(* PLC project Unnamed, Unknown Unnamed 1 *)
(* stored: creationDateTime 2023-03-29T00:03:16, modificationDateTime 2023-04-16T13:55:39 *)

PROGRAM Master_Program
  VAR
    Panel_Mag_Sensor AT %IX0.0 : BOOL;  (* Physcial Inputs on the Right Demostration Panel offset 4 input *)
    Panel_IR_Sensor AT %IX0.1 : BOOL;  (* Physcial Inputs on the Right Demostration Panel offset 6 input *)
    Panel_Motion_Sensor AT %IX0.2 : BOOL;  (* Physcial Inputs on the Right Demostration Panel offset 5 input *)
    Panel_GD_Remote_UP_PB AT %IX0.3 : BOOL;  (* Physcial Inputs on the Right Demostration Panel offset 7 input *)
    Panel_GD_Remote_DOWN_PB AT %IX0.4 : BOOL;  (* Physcial Inputs on the Right Demostration Panel offset 8 input *)
    Panel_FD_Lock_Signal AT %IX0.5 : BOOL;  (* Physcial Inputs on the Right Demostration Panel offset 9 input *)
    Panel_Arm_Panel_PB AT %IX0.6 : BOOL;  (* Physcial Inputs on the Right Demostration Panel offset 2 input *)
    Panel_Arm_House_PB AT %IX0.7 : BOOL;  (* Physcial Inputs on the Right Demostration Panel offset 3 input *)
    Panel_Reset_PB AT %IX1.0 : BOOL;  (* Physcial Inputs on the Right Demostration Panel offset 11 input *)
    Panel_FD_Unlock_Signal AT %IX1.1 : BOOL;  (* Physcial Inputs on the Right Demostration Panel offset 10 input *)
    Panel_Alarm_Light AT %QX0.0 : BOOL;  (* Alarm flashes when triggered offset 0 coil "Changed from 0.0 for testing" 102.3 for uno pin 13 *)
    Home_GD_Postion_Switch AT %IX102.0 : BOOL;  (* Physcial Inputs in the House Model offset 801 input *)
    Home_Mag_Sensor AT %IX102.1 : BOOL;  (* Physcial Inputs in the House Model offset 802 input *)
    Home_Motion_Sensor AT %IX102.2 : BOOL;  (* Physcial Inputs in the House Model offset 803 input *)
    Home_IR_Sensor AT %IX102.3 : BOOL;  (* Physcial Inputs in the House Model offset 804 input *)
    Home_Green_PB_Floor_01 AT %IX102.4 : BOOL;  (* Physcial Inputs in the House Model offset 805 input *)
    Home_Green_PB_Floor_02 AT %IX102.5 : BOOL;  (* Physcial Inputs in the House Model offset 806 input *)
    Home_Blue_PB_Floor_03 AT %IX102.6 : BOOL;  (* Physcial Inputs in the House Model offset 807 input *)
    Home_Red_PB_Floor_03 AT %IX102.7 : BOOL;  (* Physcial Inputs in the House Model offset 807 input *)
    Home_Green_LED_Floor_01 AT %QX100.0 : BOOL;  (* Digital output to control GD Motor offset 800 coil "Changed from 100.0 for testing" *)
    Home_Green_LED_Floor_02 AT %QX100.1 : BOOL;  (* Digital output to control GD Motor offset 801 coil *)
    Home_Green_LED_Floor_03 AT %QX100.2 : BOOL;  (* Digital output to control GD Motor offset 802 coil *)
    Home_White_LED_Floor_01 AT %QX100.3 : BOOL;  (* Digital output to control GD Motor offset 803 coil *)
    Home_White_LED_Floor_02 AT %QX100.4 : BOOL;  (* Digital output to control GD Motor offset 804 coil *)
    Home_White_LED_Floor_03 AT %QX100.5 : BOOL;  (* Digital output to control GD Motor offset 805 coil *)
    Home_White_LED_Floor_Backside AT %QX100.6 : BOOL;  (* Digital output to control GD Motor offset 806 coil *)
    Home_GD_Motor_UP AT %QX100.7 : BOOL;  (* Digital output to control GD Motor offset 807 coil *)
    Home_GD_Motor_DOWN AT %QX101.0 : BOOL;  (* Digital output to control GD Motor offset 808 coil *)
    Home_FD_Deadbolt AT %QX101.1 : BOOL;  (* Digital output to control FD Solenoid offset 809 coil *)
    Home_GD_Position AT %QX101.2 : BOOL;  (* Digital output to control GD Motor offset 810 coil *)
    Panel_Arm_Virtual_PB AT %QX10.0 : BOOL;  (* Virutal Push Button for HMI and attacks offset 80 coil *)
    Panel_Arm_Mag_Sensor_Virtual AT %QX10.1 : BOOL;  (* Virutal Push Button for HMI and attacks offset 81 coil *)
    Panel_Arm_Motion_Sensor_Virtual AT %QX10.2 : BOOL;  (* Virutal Push Button for HMI and attacks offset 82 coil *)
    Panel_Arm_IR_Sensor_Virtual AT %QX10.3 : BOOL;  (* Virutal Push Button for HMI and attacks offset 83 coil *)
    Panel_Mag_Sensor_Virtual AT %QX10.4 : BOOL;  (* Virutal Push Button for HMI and attacks offset 84 coil *)
    Panel_Motion_Sensor_Virtual AT %QX10.5 : BOOL;  (* Virutal Push Button for HMI and attacks offset 85 coil *)
    Panel_IR_Sensor_Virtual AT %QX10.6 : BOOL;  (* Virutal Push Button for HMI and attacks offset 86 coil *)
    Panel_GD_Up_OnOff_Virtual_PB AT %QX10.7 : BOOL;  (* Virutal Push Button for HMI and attacks offset 87 coil *)
    Panel_GD_Remote_Up_Virtual AT %QX11.0 : BOOL;  (* Virutal Push Button for HMI and attacks offset 88 coil *)
    Panel_GD_Down_OnOff_Virtual_PB AT %QX11.1 : BOOL;  (* Virutal Push Button for HMI and attacks offset 89 coil *)
    Panel_GD_Remote_Down_Virtual AT %QX11.2 : BOOL;  (* Virutal Push Button for HMI and attacks offset 90 coil *)
    Panel_FD_Lock_OnOff_Virtual_PB AT %QX11.3 : BOOL;  (* Virutal Push Button for HMI and attacks offset 91 coil *)
    Panel_FD_Lock_Signal_Virtual AT %QX11.4 : BOOL;  (* Virutal Push Button for HMI and attacks offset 92 coil *)
    Panel_FD_Unlock_OnOff_Virtual_PB AT %QX11.5 : BOOL;  (* Virutal Push Button for HMI and attacks offset 93 coil *)
    Panel_FD_Unlock_Signal_Virtual AT %QX11.6 : BOOL;  (* Virutal Push Button for HMI and attacks offset 94 coil *)
    Home_FD_Lock_Signal_Virtual AT %QX110.0 : BOOL;  (* Virutal Push Button for HMI and attacks offset 880 coil *)
    Home_FD_Unlock_Signal_Virtual AT %QX110.1 : BOOL;  (* Virutal Push Button for HMI and attacks offset 881 coil *)
    Home_Arm_Virtual_PB AT %QX110.2 : BOOL;  (* Virutal Push Button for HMI and attacks offset 882 coil *)
    Home_Arm_Mag_Sensor_Virtual AT %QX110.3 : BOOL;  (* Virutal Push Button for HMI and attacks offset 883 coil *)
    Home_Mag_Sensor_Virtual AT %QX110.4 : BOOL;  (* Virutal Push Button for HMI and attacks offset 884 coil *)
    Home_Arm_Motion_Sensor_Virtual AT %QX110.5 : BOOL;  (* Virutal Push Button for HMI and attacks offset 885 coil *)
    Home_Motion_Sensor_Virtual AT %QX110.6 : BOOL;  (* Virutal Push Button for HMI and attacks offset 886 coil *)
    Home_Arm_IR_Sensor_Virtual AT %QX110.7 : BOOL;  (* Virutal Push Button for HMI and attacks offset 887 coil *)
    Home_IR_Sensor_Virtual AT %QX111.0 : BOOL;  (* Virutal Push Button for HMI and attacks offset 888 coil *)
    Home_Green_PB_Auto_01 AT %QX111.2 : BOOL;  (* Virutal Push Button for HMI and attacks offset 890 coil *)
    Home_Green_PB_Auto_02 AT %QX111.4 : BOOL;  (* Virutal Push Button for HMI and attacks offset 892 coil *)
    Home_Green_PB_Auto_03 AT %QX111.6 : BOOL;  (* Virutal Push Button for HMI and attacks offset 894 coil *)
    Home_Green_LED_Reset_PB AT %QX111.7 : BOOL;  (* Virutal Push Button for HMI and attacks offset 895 coil *)
    Reset_Green_Lights AT %QX112.0 : BOOL;  (* Virutal Push Button for HMI and attacks offset 896 coil *)
  END_VAR
  VAR
    TON0 : TON;  (* Waits set number of seconds before reseting the green lights. *)
  END_VAR
  VAR
    Home_White_PD_Floor_01 AT %QX112.1 : BOOL;  (* Virutal Push Button for HMI and attacks offset 897 coil *)
    Home_White_PD_Floor_02 AT %QX112.2 : BOOL;  (* Virutal Push Button for HMI and attacks offset 898 coil *)
    Home_White_PD_Floor_03 AT %QX112.3 : BOOL;  (* Virutal Push Button for HMI and attacks offset 899 coil *)
    Home_White_PD_Backside AT %QX112.4 : BOOL;  (* Virutal Push Button for HMI and attacks offset 900 *)
    Home_Reset_PB_Virtual AT %QX112.5 : BOOL;  (* Virutal Push Button for HMI and attacks offset 901 *)
    Home_GD_OpenClose_Switch_Vir AT %QX112.6 : BOOL;  (* Virutal Push Button for HMI and attacks offset 902 "Testing" *)
  END_VAR

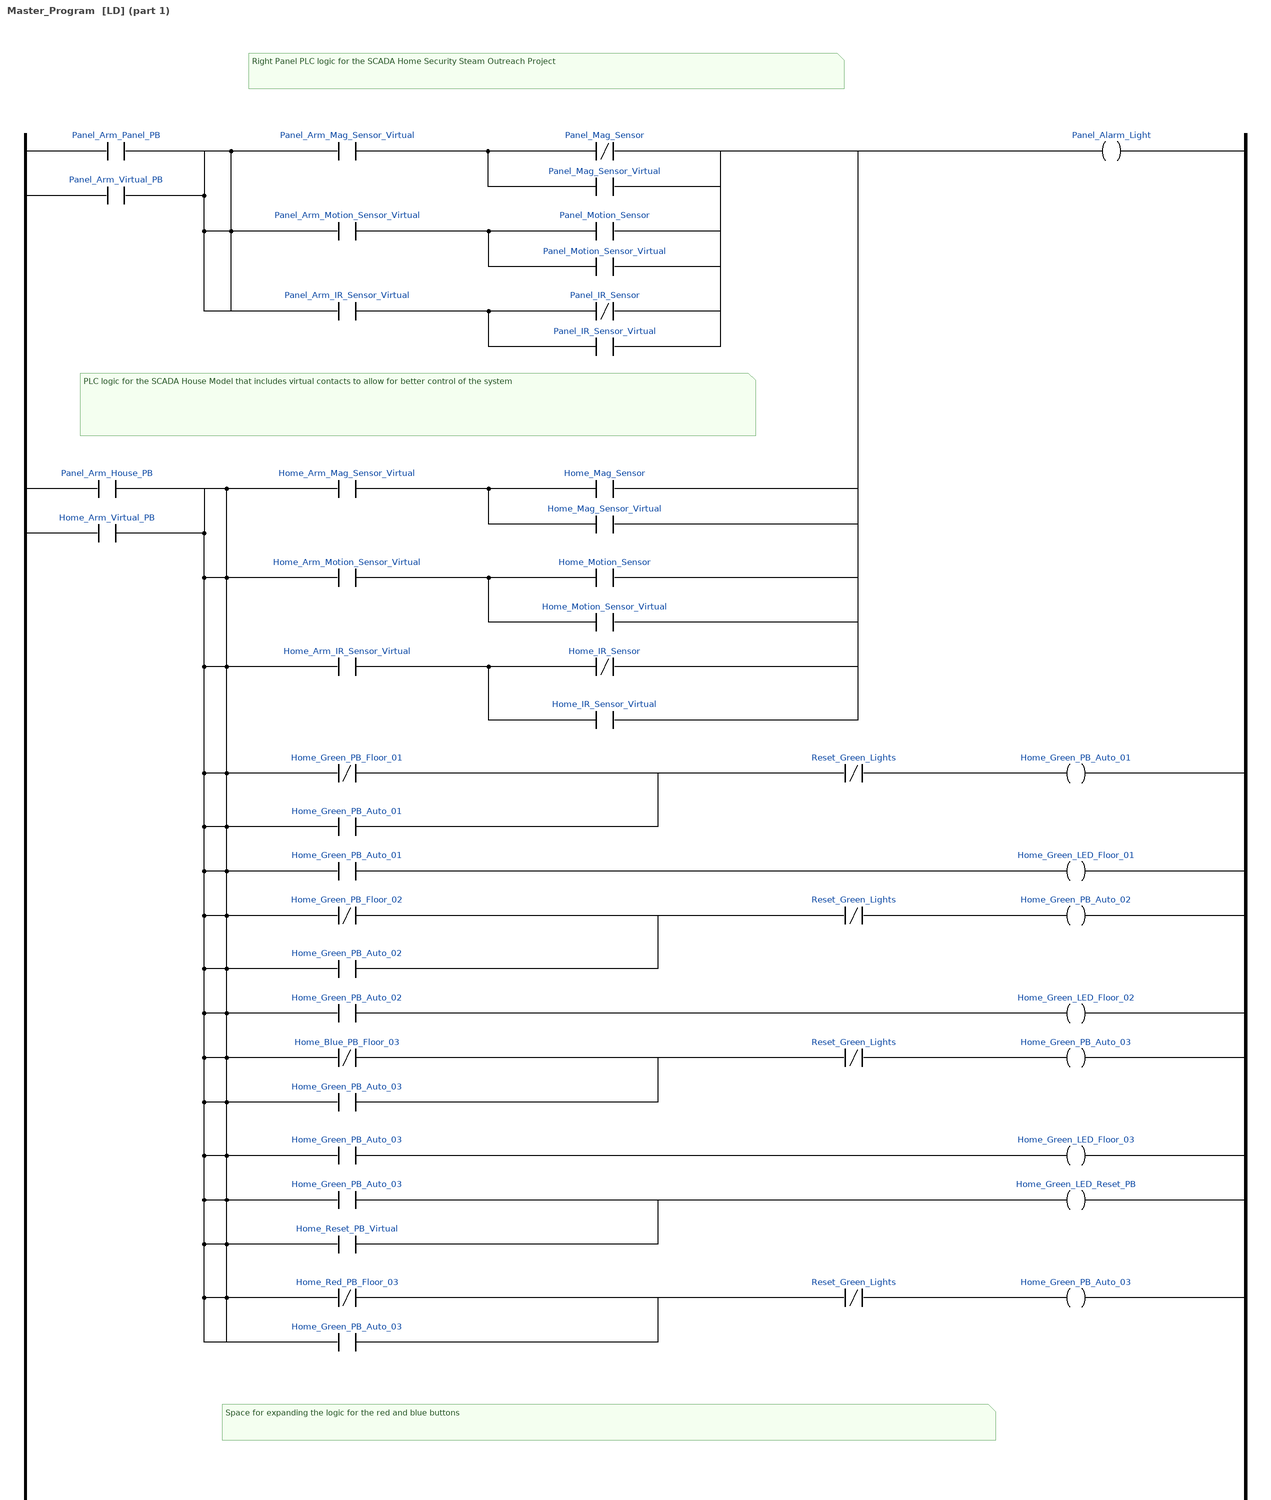
(* LD diagram, written out as Structured Text *)
(* Right Panel PLC logic for the SCADA Home Security Steam Outreach Project *)
Panel_Alarm_Light := (Panel_Arm_Panel_PB OR Panel_Arm_Virtual_PB) AND Panel_Arm_Mag_Sensor_Virtual AND NOT Panel_Mag_Sensor OR (Panel_Arm_Panel_PB OR Panel_Arm_Virtual_PB) AND Panel_Arm_Mag_Sensor_Virtual AND Panel_Mag_Sensor_Virtual OR (Panel_Arm_Panel_PB OR Panel_Arm_Virtual_PB) AND Panel_Arm_Motion_Sensor_Virtual AND Panel_Motion_Sensor OR (Panel_Arm_Panel_PB OR Panel_Arm_Virtual_PB) AND Panel_Arm_Motion_Sensor_Virtual AND Panel_Motion_Sensor_Virtual OR (Panel_Arm_Panel_PB OR Panel_Arm_Virtual_PB) AND Panel_Arm_IR_Sensor_Virtual AND NOT Panel_IR_Sensor OR (Panel_Arm_Panel_PB OR Panel_Arm_Virtual_PB) AND Panel_Arm_IR_Sensor_Virtual AND Panel_IR_Sensor_Virtual OR (Home_Arm_Virtual_PB OR Panel_Arm_House_PB) AND Home_Arm_Mag_Sensor_Virtual AND Home_Mag_Sensor OR (Home_Arm_Virtual_PB OR Panel_Arm_House_PB) AND Home_Arm_Mag_Sensor_Virtual AND Home_Mag_Sensor_Virtual OR (Home_Arm_Virtual_PB OR Panel_Arm_House_PB) AND Home_Arm_Motion_Sensor_Virtual AND Home_Motion_Sensor OR (Home_Arm_Virtual_PB OR Panel_Arm_House_PB) AND Home_Arm_Motion_Sensor_Virtual AND Home_Motion_Sensor_Virtual OR (Home_Arm_Virtual_PB OR Panel_Arm_House_PB) AND Home_Arm_IR_Sensor_Virtual AND NOT Home_IR_Sensor OR (Home_Arm_Virtual_PB OR Panel_Arm_House_PB) AND Home_Arm_IR_Sensor_Virtual AND Home_IR_Sensor_Virtual;
(* PLC logic for the SCADA House Model that includes virtual contacts to allow for better control of the system *)
Home_Green_PB_Auto_01 := (Panel_Arm_House_PB OR Home_Arm_Virtual_PB) AND (Home_Green_PB_Auto_01 OR NOT Home_Green_PB_Floor_01) AND NOT Reset_Green_Lights;
Home_Green_LED_Floor_01 := (Panel_Arm_House_PB OR Home_Arm_Virtual_PB) AND Home_Green_PB_Auto_01;
Home_Green_PB_Auto_02 := (Home_Arm_Virtual_PB OR Panel_Arm_House_PB) AND (Home_Green_PB_Auto_02 OR NOT Home_Green_PB_Floor_02) AND NOT Reset_Green_Lights;
Home_Green_LED_Floor_02 := (Home_Arm_Virtual_PB OR Panel_Arm_House_PB) AND Home_Green_PB_Auto_02;
Home_Green_PB_Auto_03 := (Home_Arm_Virtual_PB OR Panel_Arm_House_PB) AND (Home_Green_PB_Auto_03 OR NOT Home_Blue_PB_Floor_03) AND NOT Reset_Green_Lights;
Home_Green_LED_Floor_03 := (Home_Arm_Virtual_PB OR Panel_Arm_House_PB) AND Home_Green_PB_Auto_03;
Home_Green_LED_Reset_PB := (Home_Arm_Virtual_PB OR Panel_Arm_House_PB) AND (Home_Green_PB_Auto_03 OR Home_Reset_PB_Virtual);
Home_Green_PB_Auto_03 := (Panel_Arm_House_PB OR Home_Arm_Virtual_PB) AND (NOT Home_Red_PB_Floor_03 OR Home_Green_PB_Auto_03) AND NOT Reset_Green_Lights;
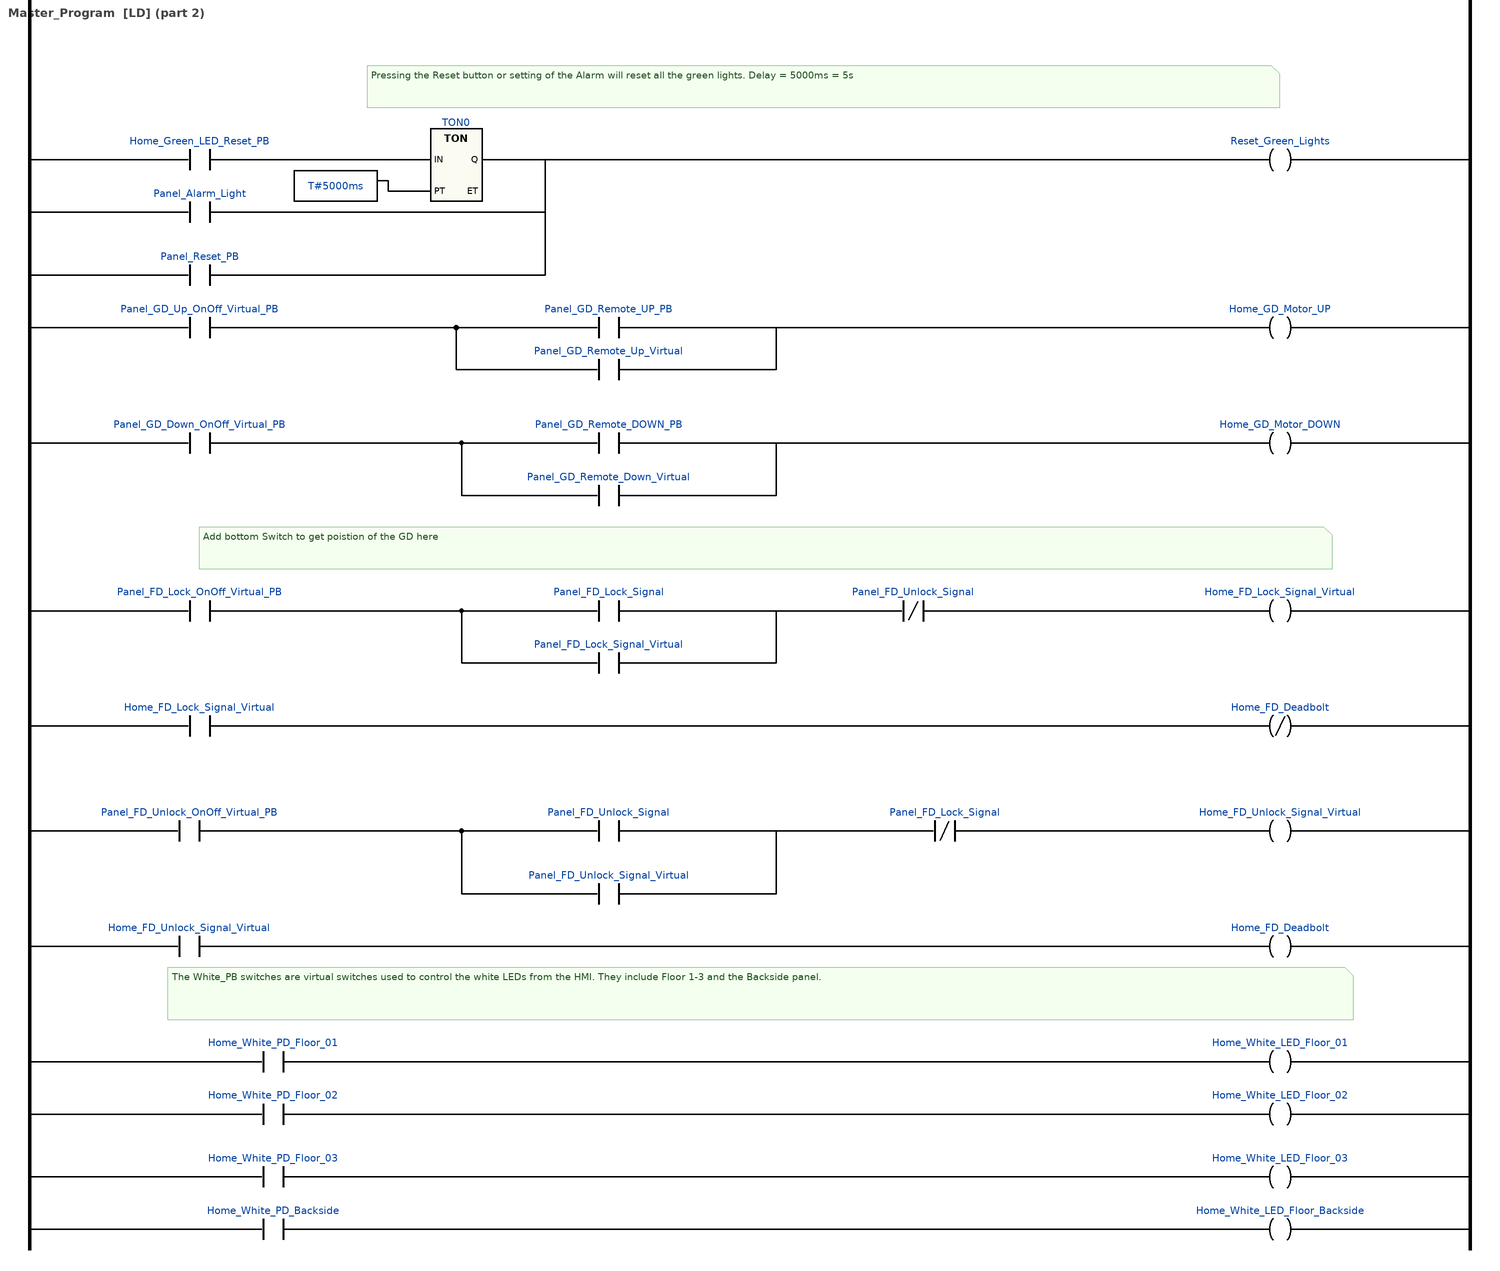
(* Space for expanding the logic for the red and blue buttons *)
(* Pressing the Reset button or setting of the Alarm will reset all the green lights. Delay = 5000ms = 5s *)
TON0(IN := Home_Green_LED_Reset_PB, PT := T#5000ms);
Reset_Green_Lights := Panel_Alarm_Light OR TON0.Q OR Panel_Reset_PB;
Home_GD_Motor_UP := Panel_GD_Up_OnOff_Virtual_PB AND (Panel_GD_Remote_UP_PB OR Panel_GD_Remote_Up_Virtual);
Home_GD_Motor_DOWN := Panel_GD_Down_OnOff_Virtual_PB AND (Panel_GD_Remote_DOWN_PB OR Panel_GD_Remote_Down_Virtual);
(* Add bottom Switch to get poistion of the GD here *)
Home_FD_Lock_Signal_Virtual := Panel_FD_Lock_OnOff_Virtual_PB AND (Panel_FD_Lock_Signal OR Panel_FD_Lock_Signal_Virtual) AND NOT Panel_FD_Unlock_Signal;
Home_FD_Deadbolt := NOT Home_FD_Lock_Signal_Virtual;
Home_FD_Unlock_Signal_Virtual := Panel_FD_Unlock_OnOff_Virtual_PB AND (Panel_FD_Unlock_Signal OR Panel_FD_Unlock_Signal_Virtual) AND NOT Panel_FD_Lock_Signal;
Home_FD_Deadbolt := Home_FD_Unlock_Signal_Virtual;
(* The White_PB switches are virtual switches used to control the white LEDs from the HMI. They include Floor 1-3 and the Backside panel. *)
Home_White_LED_Floor_01 := Home_White_PD_Floor_01;
Home_White_LED_Floor_02 := Home_White_PD_Floor_02;
Home_White_LED_Floor_03 := Home_White_PD_Floor_03;
Home_White_LED_Floor_Backside := Home_White_PD_Backside;
END_PROGRAM

CONFIGURATION Config0
  RESOURCE Res0 ON PLC
    TASK task0(INTERVAL := T#20ms, PRIORITY := 0);
    PROGRAM instance0 WITH task0 : Master_Program;
  END_RESOURCE
END_CONFIGURATION
